# B&R Automation Studio project RobotVirkNu
Automation Studio 4.3.3.196

## Configuration Config1

### Hardware
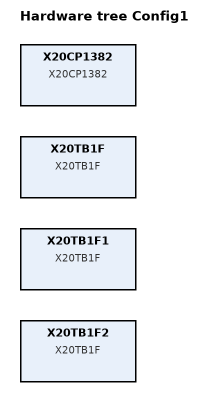
```
X20CP1382 : X20CP1382 v1.3.2.0  [X1 -> X1.SL; X2 -> X2.SL; X3 -> X3.SL]
  Module X1 (Type=X1, Virtual=true, Version=1.3.2.0)
    Connection (Connector=SS1, TargetModule=X20TB1F, TargetConnector=SS)
    Connection (Connector=SL, TargetModule=X20CP1382, TargetConnector=X1)
  Module X2 (Type=X2, Virtual=true, Version=1.3.2.0)
    Connection (Connector=SS1, TargetModule=X20TB1F1, TargetConnector=SS)
    Connection (Connector=SL, TargetModule=X20CP1382, TargetConnector=X2)
  Module X3 (Type=X3, Virtual=true, Version=1.3.2.0)
    Connection (Connector=SS1, TargetModule=X20TB1F2, TargetConnector=SS)
    Connection (Connector=SL, TargetModule=X20CP1382, TargetConnector=X3)
  Connector IF2:
    ActivateDevice = 1
  ConfigurationID = RobotVirkNu_Config1
  Simulation = 1
X20TB1F : X20TB1F v1.0.0.0
X20TB1F1 : X20TB1F v1.0.0.0
X20TB1F2 : X20TB1F v1.0.0.0
```

## Logical view

Binary libraries used (declarations not repeated): astime, operator


### Program Logical/Program (IEC)

#### Variables.var
```iecst
VAR
	commandText : STRING[20];
	i : USINT;
	input : STRING[40000];
	stepCount : USINT;
	step_timer : TON;
	test : USINT;
	timer : TON;
	x_dir : BOOL;
	x_en : BOOL;
	x_step : BOOL;
	y_dir : BOOL;
	y_en : BOOL;
	y_step : BOOL;
	z_dir : BOOL;
	z_en : BOOL;
	z_step : BOOL;
END_VAR
```

#### Main.st
```iecst
PROGRAM _INIT
	input := 'MDUMMMMMDUMMMMMDUMDUMDUMDUMDUMMMMMMMMMMMMMMDUMDUMDUMDUMDUMDUMDUMDUMDUMDUMDUMDUMMMMMMMMM';
	x_step := FALSE;
	y_step := FALSE;
	z_step := FALSE;
	x_dir := FALSE;
	y_dir := FALSE;
	z_dir := FALSE;
	x_en := TRUE;
	y_en := TRUE;
	z_en := TRUE;

	//	M = MOVE
	//	D = Down
	//	U = Up
	//	N = New line
	//	S = Sharpener

END_PROGRAM

PROGRAM _CYCLIC
	timer.IN := TRUE;
	timer.PT := T#500ms;
	step_timer.IN := FALSE;
	step_timer.PT := T#100ms;

	IF timer.Q THEN

		IF i < LEN(input) THEN
			//Change commandText to show the current function
			commandText := MID(input, 1, i);
			i := i + 1;

			WHILE commandText = 'M' AND timer.Q DO
				x_dir := TRUE;
				y_step := FALSE;
				z_step := FALSE;

				IF x_step = FALSE THEN
					x_step := TRUE;
				ELSE
					x_step := FALSE;
				END_IF

//				IF stepCount < 100 THEN
//					IF x_step = FALSE THEN
//						x_step := TRUE;
//					ELSE
//						x_step := FALSE;
//						stepCount := stepCount + 1;
//						END_IF
//
//
//				END_IF

//				//Code to move
//			ELSIF(MID(input, 1, i) = 'D') THEN
//				test := 2;
//				//Code to make the robot move down
//			ELSIF(MID(input, 1, i) = 'U') THEN
//				test := 3;
//				//Code to make the robot move up
//			ELSIF(MID(input, 1, i) = 'N') THEN
//				test := 4;
//				//Code to make the robot go to the next line
//			ELSIF(MID(input, 1, i) = 'S') THEN
//				test := 5;
//				//Code to make the robot go to the sharpener
				//
			END_WHILE
			END_IF
		timer.IN := FALSE;
	END_IF

	//Calling timer function block
	timer();

END_PROGRAM

PROGRAM _EXIT

END_PROGRAM
```

Listed in the project but not available here: Logical/Global.typ, Logical/Global.var
